PROGRAM Slits
VAR
    slitTest : FB_SlitPairV2();
END_VAR

slitTest(nIdPositiveAxis:=1, nIdNegativeAxis:=2, nIdGapSizeAxis:=3, nIdGapCentreAxis:=4, bEnable:= TRUE);

END_PROGRAM

(* stored: Version 1.1.0.1, ProductVersion 3.1.4024.11
   POU Slits: Id {f77a44d6-02e8-441c-8fcf-819361deb1ce}, SpecialFunc None *)
